TYPE "Motor2Ctrl"
VERSION : 0.1
// Block: Motor2Ctrl
   STRUCT
      SafeStop : Bool;
      Rst : Bool;
      RunBkw : Bool;
      RunFwd : Bool;
   END_STRUCT;

END_TYPE
